{attribute 'qualified_only'}
{attribute 'to_string'}
TYPE E_GCSingleProcessAxis :
(
	None := 0,
	SpinAxis := 1,
	LiftPinAxis := 2,
	Both := 3
) UINT;
END_TYPE

(* stored: Version 1.1.0.1, ProductVersion 3.1.4026.18
   DUT E_GCSingleProcessAxis: Id {d343cc97-b1b7-48f8-b368-325d48269d20} *)
